// TIA Portal V17 export
// export: Created 2024-06-14T09:53:51.024025Z, ExportSetting WithDefaults, DisplayName Totally Integrated Automation Portal, DisplayVersion V17, DisplayName TIA Portal Openness, DisplayVersion V17, DisplayName TIA Portal Version Control Interface, DisplayVersion V17, DisplayName Simotion SCOUT TIA, DisplayVersion 5.4.3.0, DisplayName SINAMICS Startdrive Advanced, DisplayVersion V17 SP1 Update 1, DisplayName SINAMICS Startdrive G110M, G120, G120C, G120D, G120P, G115D, DisplayVersion V17 SP1 Update 1, DisplayName SINAMICS Startdrive G130, G150, S120, S150, SINAMICS MV, S210, DisplayVersion V17 SP1 Update 1, DisplayName STEP 7 Professional, DisplayVersion V17, DisplayName STEP 7 Safety, DisplayVersion V17, DisplayName WinCC Professional, DisplayVersion V17
TYPE "ufinefill_station"
// stored: IsFailsafeCompliant false
   STRUCT
      INxNear_Filter_Stopper_L1 : Bool;
      INxFilling_Unit_L2 : Bool;
      INxFilling_Unit_L3 : Bool;
      INxFilling_Unit_L4 : Bool;
      INxFilling_Unit_L5 : Bool;
      INxDown_Line_Conveyor_L6 : Bool;
      INxCylinder_Selection_2 : Bool;
      INxCylinder_Selection_3 : Bool;
      INxCylinder_Selection_4 : Bool;
      INxStopper_Bypass_L2 : Bool;
      INxStopper_Bypass_L3 : Bool;
      INxStopper_Bypass_L4 : Bool;
      OUTxSolenoid_Control_Stopper_L1 : Bool;
      OUTxSolenoid_Control_LiftTable_L2 : Bool;
      OUTxSolenoid_Control_LiftTable_L3 : Bool;
      OUTxSolenoid_Control_LiftTable_L4 : Bool;
      OUTxSolenoid_Control_LiftTable_L5 : Bool;
      iSensingTime : Time;
      OUTxCylinder_Indicator_2 : Bool;
      OUTxCylinder_Indicator_3 : Bool;
      OUTxCylinder_Indicator_4 : Bool;
   END_STRUCT;
END_TYPE
